{attribute 'pack_mode' := '0'}
TYPE ST_PLCInputs :
STRUCT
	I0: BYTE;
	I1: BYTE;
	I2: BYTE;
	I3: BYTE;
	I4: BYTE;
	I5: BYTE;
	I6: BYTE;
	I7: BYTE;
	I8: BYTE;
	I9: BYTE;
	I10: BYTE;
	I11: BYTE;
	I12: BYTE;
	I13: BYTE;
	I14: BYTE;
	I15: BYTE;
	I16: BYTE;
	I17: BYTE;
	I18: BYTE;
	I19: BYTE;
	I20: BYTE;
	I21: BYTE;
	I22: BYTE;
	I23: BYTE;
	I24: BYTE;
	I25: BYTE;
	I26: BYTE;
	I27: BYTE;
	I28: BYTE;
	I29: BYTE;
	I30: BYTE;
	I31: BYTE;
	I32: BYTE;
	I33: BYTE;
	I34: BYTE;
	I35: BYTE;
	I36: BYTE;
	I37: BYTE;
	I38: BYTE;
	I39: BYTE;
	I40: BYTE;
	I41: BYTE;
	I42: BYTE;
	I43: BYTE;
	I44: BYTE;
	I45: BYTE;
	I46: BYTE;
	I47: BYTE;
	I48: BYTE;
	I49: BYTE;
	I50: BYTE;
	I51: BYTE;
	I52: BYTE;
	I53: BYTE;
	I54: BYTE;
	I55: BYTE;
	I56: BYTE;
	I57: BYTE;
	I58: BYTE;
	I59: BYTE;
	I60: BYTE;
	I61: BYTE;
	I62: BYTE;
	I63: BYTE;
	I64: BYTE;
	I65: BYTE;
	I66: BYTE;
	I67: BYTE;
	I68: BYTE;
	I69: BYTE;
	I70: BYTE;
	I71: BYTE;
	I72: BYTE;
	I73: BYTE;
	I74: BYTE;
	I75: BYTE;
	I76: BYTE;
	I77: BYTE;
	I78: BYTE;
	I79: BYTE;
	I80: BYTE;
	I81: BYTE;
	I82: BYTE;
	I83: BYTE;
	I84: BYTE;
	I85: BYTE;
	I86: BYTE;
	I87: BYTE;
	I88: BYTE;
	I89: BYTE;
	I90: BYTE;
	I91: BYTE;
	I92: BYTE;
	I93: BYTE;
	I94: BYTE;
	I95: BYTE;
	I96: BYTE;
	I97: BYTE;
	I98: BYTE;
	I99: BYTE;
	I100: BYTE;
	I101: BYTE;
	I102: BYTE;
	I103: BYTE;
	I104: BYTE;
	I105: BYTE;
	I106: BYTE;
	I107: BYTE;
	I108: BYTE;
	I109: BYTE;
	I110: BYTE;
	I111: BYTE;
	I112: BYTE;
	I113: BYTE;
	I114: BYTE;
	I115: BYTE;
	I116: BYTE;
	I117: BYTE;
	I118: BYTE;
	I119: BYTE;
	I120: BYTE;
	I121: BYTE;
	I122: BYTE;
	I123: BYTE;
	I124: BYTE;
	I125: BYTE;
	I126: BYTE;
	I127: BYTE;
	I128: BYTE;
	I129: BYTE;
	I130: BYTE;
	I131: BYTE;
	I132: BYTE;
	I133: BYTE;
	I134: BYTE;
	I135: BYTE;
	I136: BYTE;
	I137: BYTE;
	I138: BYTE;
	I139: BYTE;
	I140: BYTE;
	I141: BYTE;
	I142: BYTE;
	I143: BYTE;
	I144: BYTE;
	I145: BYTE;
	I146: BYTE;
	I147: BYTE;
	I148: BYTE;
	I149: BYTE;
	I150: BYTE;
	I151: BYTE;
	I152: BYTE;
	I153: BYTE;
	I154: BYTE;
	I155: BYTE;
	I156: BYTE;
	I157: BYTE;
	I158: BYTE;
	I159: BYTE;
	I160: BYTE;
	I161: BYTE;
	I162: BYTE;
	I163: BYTE;
	I164: BYTE;
	I165: BYTE;
	I166: BYTE;
	I167: BYTE;
	I168: BYTE;
	I169: BYTE;
	I170: BYTE;
	I171: BYTE;
	I172: BYTE;
	I173: BYTE;
	I174: BYTE;
	I175: BYTE;
	I176: BYTE;
	I177: BYTE;
	I178: BYTE;
	I179: BYTE;
	I180: BYTE;
	I181: BYTE;
	I182: BYTE;
	I183: BYTE;
	I184: BYTE;
	I185: BYTE;
	I186: BYTE;
	I187: BYTE;
	I188: BYTE;
	I189: BYTE;
	I190: BYTE;
	I191: BYTE;
	I192: BYTE;
	I193: BYTE;
	I194: BYTE;
	I195: BYTE;
	I196: BYTE;
	I197: BYTE;
	I198: BYTE;
	I199: BYTE;
	I200: BYTE;
	I201: BYTE;
	I202: BYTE;
	I203: BYTE;
	I204: BYTE;
	I205: BYTE;
	I206: BYTE;
	I207: BYTE;
	I208: BYTE;
	I209: BYTE;
	I210: BYTE;
	I211: BYTE;
	I212: BYTE;
	I213: BYTE;
	I214: BYTE;
	I215: BYTE;
	I216: BYTE;
	I217: BYTE;
	I218: BYTE;
	I219: BYTE;
	I220: BYTE;
	I221: BYTE;
	I222: BYTE;
	I223: BYTE;
	I224: BYTE;
	I225: BYTE;
	I226: BYTE;
	I227: BYTE;
	I228: BYTE;
	I229: BYTE;
	I230: BYTE;
	I231: BYTE;
	I232: BYTE;
	I233: BYTE;
	I234: BYTE;
	I235: BYTE;
	I236: BYTE;
	I237: BYTE;
	I238: BYTE;
	I239: BYTE;
	I240: BYTE;
	I241: BYTE;
	I242: BYTE;
	I243: BYTE;
	I244: BYTE;
	I245: BYTE;
	I246: BYTE;
	I247: BYTE;
	I248: BYTE;
	I249: BYTE;
	I250: BYTE;
	I251: BYTE;
	I252: BYTE;
	I253: BYTE;
	I254: BYTE;
	I255: BYTE;
	I256: BYTE;
	I257: BYTE;
	I258: BYTE;
	I259: BYTE;
	I260: BYTE;
	I261: BYTE;
	I262: BYTE;
	I263: BYTE;
	I264: BYTE;
	I265: BYTE;
	I266: BYTE;
	I267: BYTE;
	I268: BYTE;
	I269: BYTE;
	I270: BYTE;
	I271: BYTE;
	I272: BYTE;
	I273: BYTE;
	I274: BYTE;
	I275: BYTE;
	I276: BYTE;
	I277: BYTE;
	I278: BYTE;
	I279: BYTE;
	I280: BYTE;
	I281: BYTE;
	I282: BYTE;
	I283: BYTE;
	I284: BYTE;
	I285: BYTE;
	I286: BYTE;
	I287: BYTE;
	I288: BYTE;
	I289: BYTE;
	I290: BYTE;
	I291: BYTE;
	I292: BYTE;
	I293: BYTE;
	I294: BYTE;
	I295: BYTE;
	I296: BYTE;
	I297: BYTE;
	I298: BYTE;
	I299: BYTE;
	I300: BYTE;
	I301: BYTE;
	I302: BYTE;
	I303: BYTE;
	I304: BYTE;
	I305: BYTE;
	I306: BYTE;
	I307: BYTE;
	I308: BYTE;
	I309: BYTE;
	I310: BYTE;
	I311: BYTE;
	I312: BYTE;
	I313: BYTE;
	I314: BYTE;
	I315: BYTE;
	I316: BYTE;
	I317: BYTE;
	I318: BYTE;
	I319: BYTE;
	I320: BYTE;
	I321: BYTE;
	I322: BYTE;
	I323: BYTE;
	I324: BYTE;
	I325: BYTE;
	I326: BYTE;
	I327: BYTE;
	I328: BYTE;
	I329: BYTE;
	I330: BYTE;
	I331: BYTE;
	I332: BYTE;
	I333: BYTE;
	I334: BYTE;
	I335: BYTE;
	I336: BYTE;
	I337: BYTE;
	I338: BYTE;
	I339: BYTE;
	I340: BYTE;
	I341: BYTE;
	I342: BYTE;
	I343: BYTE;
	I344: BYTE;
	I345: BYTE;
	I346: BYTE;
	I347: BYTE;
	I348: BYTE;
	I349: BYTE;
	I350: BYTE;
	I351: BYTE;
	I352: BYTE;
	I353: BYTE;
	I354: BYTE;
	I355: BYTE;
	I356: BYTE;
	I357: BYTE;
	I358: BYTE;
	I359: BYTE;
	I360: BYTE;
	I361: BYTE;
	I362: BYTE;
	I363: BYTE;
	I364: BYTE;
	I365: BYTE;
	I366: BYTE;
	I367: BYTE;
	I368: BYTE;
	I369: BYTE;
	I370: BYTE;
	I371: BYTE;
	I372: BYTE;
	I373: BYTE;
	I374: BYTE;
	I375: BYTE;
	I376: BYTE;
	I377: BYTE;
	I378: BYTE;
	I379: BYTE;
	I380: BYTE;
	I381: BYTE;
	I382: BYTE;
	I383: BYTE;
	I384: BYTE;
	I385: BYTE;
	I386: BYTE;
	I387: BYTE;
	I388: BYTE;
	I389: BYTE;
	I390: BYTE;
	I391: BYTE;
	I392: BYTE;
	I393: BYTE;
	I394: BYTE;
	I395: BYTE;
	I396: BYTE;
	I397: BYTE;
	I398: BYTE;
	I399: BYTE;
	I400: BYTE;
	I401: BYTE;
	I402: BYTE;
	I403: BYTE;
	I404: BYTE;
	I405: BYTE;
	I406: BYTE;
	I407: BYTE;
	I408: BYTE;
	I409: BYTE;
	I410: BYTE;
	I411: BYTE;
	I412: BYTE;
	I413: BYTE;
	I414: BYTE;
	I415: BYTE;
	I416: BYTE;
	I417: BYTE;
	I418: BYTE;
	I419: BYTE;
	I420: BYTE;
	I421: BYTE;
	I422: BYTE;
	I423: BYTE;
	I424: BYTE;
	I425: BYTE;
	I426: BYTE;
	I427: BYTE;
	I428: BYTE;
	I429: BYTE;
	I430: BYTE;
	I431: BYTE;
	I432: BYTE;
	I433: BYTE;
	I434: BYTE;
	I435: BYTE;
	I436: BYTE;
	I437: BYTE;
	I438: BYTE;
	I439: BYTE;
	I440: BYTE;
	I441: BYTE;
	I442: BYTE;
	I443: BYTE;
	I444: BYTE;
	I445: BYTE;
	I446: BYTE;
	I447: BYTE;
	I448: BYTE;
	I449: BYTE;
	I450: BYTE;
	I451: BYTE;
	I452: BYTE;
	I453: BYTE;
	I454: BYTE;
	I455: BYTE;
	I456: BYTE;
	I457: BYTE;
	I458: BYTE;
	I459: BYTE;
	I460: BYTE;
	I461: BYTE;
	I462: BYTE;
	I463: BYTE;
	I464: BYTE;
	I465: BYTE;
	I466: BYTE;
	I467: BYTE;
	I468: BYTE;
	I469: BYTE;
	I470: BYTE;
	I471: BYTE;
	I472: BYTE;
	I473: BYTE;
	I474: BYTE;
	I475: BYTE;
	I476: BYTE;
	I477: BYTE;
	I478: BYTE;
	I479: BYTE;
	I480: BYTE;
	I481: BYTE;
	I482: BYTE;
	I483: BYTE;
	I484: BYTE;
	I485: BYTE;
	I486: BYTE;
	I487: BYTE;
	I488: BYTE;
	I489: BYTE;
	I490: BYTE;
	I491: BYTE;
	I492: BYTE;
	I493: BYTE;
	I494: BYTE;
	I495: BYTE;
	I496: BYTE;
	I497: BYTE;
	I498: BYTE;
	I499: BYTE;
	I500: BYTE;
	I501: BYTE;
	I502: BYTE;
	I503: BYTE;
	I504: BYTE;
	I505: BYTE;
	I506: BYTE;
	I507: BYTE;
	I508: BYTE;
	I509: BYTE;
	I510: BYTE;
	I511: BYTE;
	I512: BYTE;
	I513: BYTE;
	I514: BYTE;
	I515: BYTE;
	I516: BYTE;
	I517: BYTE;
	I518: BYTE;
	I519: BYTE;
	I520: BYTE;
	I521: BYTE;
	I522: BYTE;
	I523: BYTE;
	I524: BYTE;
	I525: BYTE;
	I526: BYTE;
	I527: BYTE;
	I528: BYTE;
	I529: BYTE;
	I530: BYTE;
	I531: BYTE;
	I532: BYTE;
	I533: BYTE;
	I534: BYTE;
	I535: BYTE;
	I536: BYTE;
	I537: BYTE;
	I538: BYTE;
	I539: BYTE;
	I540: BYTE;
	I541: BYTE;
	I542: BYTE;
	I543: BYTE;
	I544: BYTE;
	I545: BYTE;
	I546: BYTE;
	I547: BYTE;
	I548: BYTE;
	I549: BYTE;
	I550: BYTE;
	I551: BYTE;
	I552: BYTE;
	I553: BYTE;
	I554: BYTE;
	I555: BYTE;
	I556: BYTE;
	I557: BYTE;
	I558: BYTE;
	I559: BYTE;
	I560: BYTE;
	I561: BYTE;
	I562: BYTE;
	I563: BYTE;
	I564: BYTE;
	I565: BYTE;
	I566: BYTE;
	I567: BYTE;
	I568: BYTE;
	I569: BYTE;
	I570: BYTE;
	I571: BYTE;
	I572: BYTE;
	I573: BYTE;
	I574: BYTE;
	I575: BYTE;
	I576: BYTE;
	I577: BYTE;
	I578: BYTE;
	I579: BYTE;
	I580: BYTE;
	I581: BYTE;
	I582: BYTE;
	I583: BYTE;
	I584: BYTE;
	I585: BYTE;
	I586: BYTE;
	I587: BYTE;
	I588: BYTE;
	I589: BYTE;
	I590: BYTE;
	I591: BYTE;
	I592: BYTE;
	I593: BYTE;
	I594: BYTE;
	I595: BYTE;
	I596: BYTE;
	I597: BYTE;
	I598: BYTE;
	I599: BYTE;
	I600: BYTE;
	I601: BYTE;
	I602: BYTE;
	I603: BYTE;
	I604: BYTE;
	I605: BYTE;
	I606: BYTE;
	I607: BYTE;
	I608: BYTE;
	I609: BYTE;
	I610: BYTE;
	I611: BYTE;
	I612: BYTE;
	I613: BYTE;
	I614: BYTE;
	I615: BYTE;
	I616: BYTE;
	I617: BYTE;
	I618: BYTE;
	I619: BYTE;
	I620: BYTE;
	I621: BYTE;
	I622: BYTE;
	I623: BYTE;
	I624: BYTE;
	I625: BYTE;
	I626: BYTE;
	I627: BYTE;
	I628: BYTE;
	I629: BYTE;
	I630: BYTE;
	I631: BYTE;
	I632: BYTE;
	I633: BYTE;
	I634: BYTE;
	I635: BYTE;
	I636: BYTE;
	I637: BYTE;
	I638: BYTE;
	I639: BYTE;
	I640: BYTE;
	I641: BYTE;
	I642: BYTE;
	I643: BYTE;
	I644: BYTE;
	I645: BYTE;
	I646: BYTE;
	I647: BYTE;
	I648: BYTE;
	I649: BYTE;
	I650: BYTE;
	I651: BYTE;
	I652: BYTE;
	I653: BYTE;
	I654: BYTE;
	I655: BYTE;
	I656: BYTE;
	I657: BYTE;
	I658: BYTE;
	I659: BYTE;
	I660: BYTE;
	I661: BYTE;
	I662: BYTE;
	I663: BYTE;
	I664: BYTE;
	I665: BYTE;
	I666: BYTE;
	I667: BYTE;
	I668: BYTE;
	I669: BYTE;
	I670: BYTE;
	I671: BYTE;
	I672: BYTE;
	I673: BYTE;
	I674: BYTE;
	I675: BYTE;
	I676: BYTE;
	I677: BYTE;
	I678: BYTE;
	I679: BYTE;
	I680: BYTE;
	I681: BYTE;
	I682: BYTE;
	I683: BYTE;
	I684: BYTE;
	I685: BYTE;
	I686: BYTE;
	I687: BYTE;
	I688: BYTE;
	I689: BYTE;
	I690: BYTE;
	I691: BYTE;
	I692: BYTE;
	I693: BYTE;
	I694: BYTE;
	I695: BYTE;
	I696: BYTE;
	I697: BYTE;
	I698: BYTE;
	I699: BYTE;
	I700: BYTE;
	I701: BYTE;
	I702: BYTE;
	I703: BYTE;
	I704: BYTE;
	I705: BYTE;
	I706: BYTE;
	I707: BYTE;
	I708: BYTE;
	I709: BYTE;
	I710: BYTE;
	I711: BYTE;
	I712: BYTE;
	I713: BYTE;
	I714: BYTE;
	I715: BYTE;
	I716: BYTE;
	I717: BYTE;
	I718: BYTE;
	I719: BYTE;
	I720: BYTE;
	I721: BYTE;
	I722: BYTE;
	I723: BYTE;
	I724: BYTE;
	I725: BYTE;
	I726: BYTE;
	I727: BYTE;
	I728: BYTE;
	I729: BYTE;
	I730: BYTE;
	I731: BYTE;
	I732: BYTE;
	I733: BYTE;
	I734: BYTE;
	I735: BYTE;
	I736: BYTE;
	I737: BYTE;
	I738: BYTE;
	I739: BYTE;
	I740: BYTE;
	I741: BYTE;
	I742: BYTE;
	I743: BYTE;
	I744: BYTE;
	I745: BYTE;
	I746: BYTE;
	I747: BYTE;
	I748: BYTE;
	I749: BYTE;
	I750: BYTE;
	I751: BYTE;
	I752: BYTE;
	I753: BYTE;
	I754: BYTE;
	I755: BYTE;
	I756: BYTE;
	I757: BYTE;
	I758: BYTE;
	I759: BYTE;
	I760: BYTE;
	I761: BYTE;
	I762: BYTE;
	I763: BYTE;
	I764: BYTE;
	I765: BYTE;
	I766: BYTE;
	I767: BYTE;
	I768: BYTE;
	I769: BYTE;
	I770: BYTE;
	I771: BYTE;
	I772: BYTE;
	I773: BYTE;
	I774: BYTE;
	I775: BYTE;
	I776: BYTE;
	I777: BYTE;
	I778: BYTE;
	I779: BYTE;
	I780: BYTE;
	I781: BYTE;
	I782: BYTE;
	I783: BYTE;
	I784: BYTE;
	I785: BYTE;
	I786: BYTE;
	I787: BYTE;
	I788: BYTE;
	I789: BYTE;
	I790: BYTE;
	I791: BYTE;
	I792: BYTE;
	I793: BYTE;
	I794: BYTE;
	I795: BYTE;
	I796: BYTE;
	I797: BYTE;
	I798: BYTE;
	I799: BYTE;
	I800: BYTE;
	I801: BYTE;
	I802: BYTE;
	I803: BYTE;
	I804: BYTE;
	I805: BYTE;
	I806: BYTE;
	I807: BYTE;
	I808: BYTE;
	I809: BYTE;
	I810: BYTE;
	I811: BYTE;
	I812: BYTE;
	I813: BYTE;
	I814: BYTE;
	I815: BYTE;
	I816: BYTE;
	I817: BYTE;
	I818: BYTE;
	I819: BYTE;
	I820: BYTE;
	I821: BYTE;
	I822: BYTE;
	I823: BYTE;
	I824: BYTE;
	I825: BYTE;
	I826: BYTE;
	I827: BYTE;
	I828: BYTE;
	I829: BYTE;
	I830: BYTE;
	I831: BYTE;
	I832: BYTE;
	I833: BYTE;
	I834: BYTE;
	I835: BYTE;
	I836: BYTE;
	I837: BYTE;
	I838: BYTE;
	I839: BYTE;
	I840: BYTE;
	I841: BYTE;
	I842: BYTE;
	I843: BYTE;
	I844: BYTE;
	I845: BYTE;
	I846: BYTE;
	I847: BYTE;
	I848: BYTE;
	I849: BYTE;
	I850: BYTE;
	I851: BYTE;
	I852: BYTE;
	I853: BYTE;
	I854: BYTE;
	I855: BYTE;
	I856: BYTE;
	I857: BYTE;
	I858: BYTE;
	I859: BYTE;
	I860: BYTE;
	I861: BYTE;
	I862: BYTE;
	I863: BYTE;
	I864: BYTE;
	I865: BYTE;
	I866: BYTE;
	I867: BYTE;
	I868: BYTE;
	I869: BYTE;
	I870: BYTE;
	I871: BYTE;
	I872: BYTE;
	I873: BYTE;
	I874: BYTE;
	I875: BYTE;
	I876: BYTE;
	I877: BYTE;
	I878: BYTE;
	I879: BYTE;
	I880: BYTE;
	I881: BYTE;
	I882: BYTE;
	I883: BYTE;
	I884: BYTE;
	I885: BYTE;
	I886: BYTE;
	I887: BYTE;
	I888: BYTE;
	I889: BYTE;
	I890: BYTE;
	I891: BYTE;
	I892: BYTE;
	I893: BYTE;
	I894: BYTE;
	I895: BYTE;
	I896: BYTE;
	I897: BYTE;
	I898: BYTE;
	I899: BYTE;
	I900: BYTE;
	I901: BYTE;
	I902: BYTE;
	I903: BYTE;
	I904: BYTE;
	I905: BYTE;
	I906: BYTE;
	I907: BYTE;
	I908: BYTE;
	I909: BYTE;
	I910: BYTE;
	I911: BYTE;
	I912: BYTE;
	I913: BYTE;
	I914: BYTE;
	I915: BYTE;
	I916: BYTE;
	I917: BYTE;
	I918: BYTE;
	I919: BYTE;
	I920: BYTE;
	I921: BYTE;
	I922: BYTE;
	I923: BYTE;
	I924: BYTE;
	I925: BYTE;
	I926: BYTE;
	I927: BYTE;
	I928: BYTE;
	I929: BYTE;
	I930: BYTE;
	I931: BYTE;
	I932: BYTE;
	I933: BYTE;
	I934: BYTE;
	I935: BYTE;
	I936: BYTE;
	I937: BYTE;
	I938: BYTE;
	I939: BYTE;
	I940: BYTE;
	I941: BYTE;
	I942: BYTE;
	I943: BYTE;
	I944: BYTE;
	I945: BYTE;
	I946: BYTE;
	I947: BYTE;
	I948: BYTE;
	I949: BYTE;
	I950: BYTE;
	I951: BYTE;
	I952: BYTE;
	I953: BYTE;
	I954: BYTE;
	I955: BYTE;
	I956: BYTE;
	I957: BYTE;
	I958: BYTE;
	I959: BYTE;
	I960: BYTE;
	I961: BYTE;
	I962: BYTE;
	I963: BYTE;
	I964: BYTE;
	I965: BYTE;
	I966: BYTE;
	I967: BYTE;
	I968: BYTE;
	I969: BYTE;
	I970: BYTE;
	I971: BYTE;
	I972: BYTE;
	I973: BYTE;
	I974: BYTE;
	I975: BYTE;
	I976: BYTE;
	I977: BYTE;
	I978: BYTE;
	I979: BYTE;
	I980: BYTE;
	I981: BYTE;
	I982: BYTE;
	I983: BYTE;
	I984: BYTE;
	I985: BYTE;
	I986: BYTE;
	I987: BYTE;
	I988: BYTE;
	I989: BYTE;
	I990: BYTE;
	I991: BYTE;
	I992: BYTE;
	I993: BYTE;
	I994: BYTE;
	I995: BYTE;
	I996: BYTE;
	I997: BYTE;
	I998: BYTE;
	I999: BYTE;
	I1000: BYTE;
	I1001: BYTE;
	I1002: BYTE;
	I1003: BYTE;
	I1004: BYTE;
	I1005: BYTE;
	I1006: BYTE;
	I1007: BYTE;
	I1008: BYTE;
	I1009: BYTE;
	I1010: BYTE;
	I1011: BYTE;
	I1012: BYTE;
	I1013: BYTE;
	I1014: BYTE;
	I1015: BYTE;
	I1016: BYTE;
	I1017: BYTE;
	I1018: BYTE;
	I1019: BYTE;
	I1020: BYTE;
	I1021: BYTE;
	I1022: BYTE;
	I1023: BYTE;
END_STRUCT
END_TYPE

(* stored: Version 1.1.0.1, ProductVersion 3.1.4026.19
   DUT ST_PLCInputs: Id {52433ead-1baf-4a3d-94ba-a548f048e536} *)
